(* CoDeSys 2.3 export: JULKA.EXP *)

(* POU Rooms/Julka, ST *)
FUNCTION_BLOCK Julka
VAR
	mainLamp :OnOff;
	buttonJ8_1b: Button;
	shaderJ:Shader;
END_VAR
mainLamp(input:=J8_1a, output => J2_1);

buttonJ8_1b(input:=J8_1b);
shaderJ(switch:=buttonJ8_1b.fallingEdge);
J5_1a:=shaderJ.opening;
J5_1b:=shaderJ.closing;
END_FUNCTION_BLOCK
